# EPICS substitutions: evrSupport/Db/ioc/evrPatternXL05.substitutions
#
# Pattern records
file evrPatternAll.db {
#	    Device        ,  SLC Pattern Check LNK    , EVR/Trigger
#	                                                  Links
  pattern { DEVICE        ,        LINK4              , LINK5 , LINK6 , LINKD }
	  { IOC:XL05:EV01 ,         ""                ,  ""   ,  ""   ,  ""   }
}
file evrPatternProc.db {
  pattern { DEVICE }
	  { IOC:XL05:EV01}
}
